(* PLC project SafeLOGIC, BrAutomation SafeDESIGNER  5.24.1.0 *)
(* stored: companyURL http://www.br-automation.com, creationDateTime Sun Oct 26 13:20:25 2025 *)

PROGRAM Main

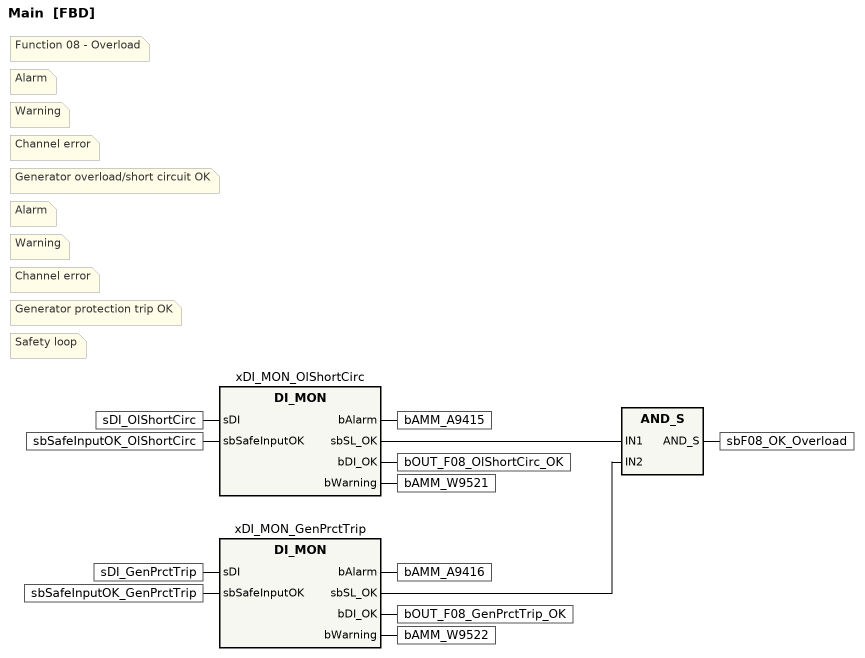
(* FBD diagram, written out as Structured Text *)
(* Function 08 - Overload *)
(* Alarm *)
xDI_MON_OlShortCirc(sDI := sDI_OlShortCirc, sbSafeInputOK := sbSafeInputOK_OlShortCirc);
bAMM_A9415 := xDI_MON_OlShortCirc.bAlarm;
(* Channel error *)
(* Generator overload/short circuit OK *)
(* Warning *)
(* Safety loop *)
bAMM_W9521 := xDI_MON_OlShortCirc.bWarning;
bOUT_F08_OlShortCirc_OK := xDI_MON_OlShortCirc.bDI_OK;
(* Alarm *)
xDI_MON_GenPrctTrip(sDI := sDI_GenPrctTrip, sbSafeInputOK := sbSafeInputOK_GenPrctTrip);
bAMM_A9416 := xDI_MON_GenPrctTrip.bAlarm;
sbF08_OK_Overload := AND_S(xDI_MON_OlShortCirc.sbSL_OK, xDI_MON_GenPrctTrip.sbSL_OK);
(* Channel error *)
(* Generator protection trip OK *)
(* Warning *)
bAMM_W9522 := xDI_MON_GenPrctTrip.bWarning;
bOUT_F08_GenPrctTrip_OK := xDI_MON_GenPrctTrip.bDI_OK;
END_PROGRAM
